PROGRAM MAIN
VAR
END_VAR

END_PROGRAM

(* stored: Version 1.1.0.1
   POU MAIN: Id {9858a2be-49fb-469e-93ec-63ca64f88c84} *)
